(* IEC 61131-3 sources: PLC-Based-Conveyor-Sorting-System/src, 2 files *)

(* ---- Main_FSM.st ---- *)
// ==============================================================================
// Conveyor Sorting System: Finite State Machine (FSM)
// Language: Structured Text (IEC 61131-3)
// ==============================================================================

PROGRAM Main_FSM
VAR
    // State Enumerations
    STATE_IDLE : INT := 1;
    STATE_RUNNING : INT := 2;
    STATE_SORTING : INT := 3;
    STATE_FAULT : INT := 4;

    Current_State : INT := STATE_IDLE;

    // Internal Flags
    b_EStop_Fault : BOOL := FALSE;
    b_Batch_Complete : BOOL := FALSE;
END_VAR

// 1. Safety & Fault Monitoring (Overrides all other logic)
IF NOT(i_EStop_Mon) THEN
    b_EStop_Fault := TRUE;
    Current_State := STATE_FAULT;
END_IF;

// 2. State Machine Transitions
CASE Current_State OF

    STATE_IDLE:
        // Transition: Idle -> Running
        IF i_Start_PB AND NOT(i_Stop_PB) AND i_EStop_Mon AND NOT(b_EStop_Fault) THEN
            Current_State := STATE_RUNNING;
        END_IF;

    STATE_RUNNING:
        // Transition: Running -> Idle (Normal Stop)
        IF i_Stop_PB THEN
            Current_State := STATE_IDLE;
        END_IF;

        // Transition: Running -> Sorting
        IF i_Prox_Sensor AND NOT(b_EStop_Fault) AND NOT(b_Batch_Complete) THEN
            Current_State := STATE_SORTING;
        END_IF;

    STATE_SORTING:
        // Transition logic back to running handled in Sorting_Logic block
        // (Ensures race conditions do not occur)

    STATE_FAULT:
        // Outputs forced to fail-safe; requires manual hardware reset
        q_Conv_Motor := FALSE;
        q_Reject_Push := FALSE;
        q_Warn_Light := TRUE;

END_CASE;

// 3. Physical Output Mapping
q_Conv_Motor := (Current_State = STATE_RUNNING) OR (Current_State = STATE_SORTING);
q_Warn_Light := (Current_State = STATE_FAULT);

END_PROGRAM

(* ---- Sorting_Logic.st ---- *)
// ==============================================================================
// Sorting Mechanics: Edge Detection & Pneumatic Transit Timing
// Language: Structured Text (IEC 61131-3)
// ==============================================================================

PROGRAM Sorting_Logic
VAR
    // Edge Detection Variables
    Prox_Previous_State : BOOL := FALSE;
    Prox_R_TRIG : BOOL := FALSE; // Rising Edge Pulse

    // Counters and Timers
    Box_Counter : CTU; // Up-Counter for Batching
    Transit_Timer : TON; // On-Delay Timer for Pneumatics
END_VAR

// 1. Positive Edge Detection (R_TRIG)
// Prevents spatial-temporal mismatch (40 false counts for 1 box)
Prox_R_TRIG := i_Prox_Sensor AND NOT(Prox_Previous_State);
Prox_Previous_State := i_Prox_Sensor;

// 2. Batch Counting
// Accumulates exactly one discrete event occurrence per physical item
Box_Counter(CU := Prox_R_TRIG, PV := 50, RESET := (Current_State = STATE_IDLE));
IF Box_Counter.Q THEN
    b_Batch_Complete := TRUE;
END_IF;

// 3. Transit Timing Physics Calculation
// Distance (d) = 0.75m | Velocity (v) = 0.5m/s | Time (t) = 1.5s
// Goal: Measures elapsed physical duration to actuate diverter accurately
Transit_Timer(
    IN := (Current_State = STATE_SORTING) AND i_Tall_Sensor,
    PT := T#1500MS // 1.5 Second precise delay
);

// Actuate Solenoid Valve
IF Transit_Timer.Q THEN
    q_Reject_Push := TRUE;
    // Reset state after sorting action
    Current_State := STATE_RUNNING;
ELSE
    q_Reject_Push := FALSE;
END_IF;

END_PROGRAM
